Staubli VAL3: table.pjx

--- table.pjx ---
Parameters version=s8.13.1Cs9_BS2800 stackSize=5000 millimeterUnit=true
Data file=table.dtx

--- table.dtx ---
mdesc mNomSpeed
public num nMatrix[1 1]
